FUNCTION_BLOCK FB_Flash
VAR_INPUT
	Input : ARRAY[0..999] OF BOOL;
	OffTime : TIME;
	OnTime :  TIME;
END_VAR
VAR_OUTPUT
	Output : ARRAY[0..999] OF BOOL;
END_VAR
VAR
	OffTimer : TON;
	OnTimer	:	TON;
	i: INT;
END_VAR

OnTimer.PT 	:= OnTime;
OffTimer.PT := OffTime;

OffTimer.IN := NOT(OnTimer.Q);
OnTimer.IN := OffTimer.Q;
		
	
FOR i := 0 TO 999 DO
	IF Input[i] THEN
		Output[i] := OnTimer.IN;
	ELSE 
		Output[i] := FALSE;
	END_IF
END_FOR
OnTimer();
OffTimer();

END_FUNCTION_BLOCK

(* stored: Version 1.1.0.1, ProductVersion 3.1.4024.12
   POU FB_Flash: Id {608cc737-8480-4ed5-9f66-37979e65114e}, SpecialFunc None *)
